// Mitsubishi GX Works2 project: Star delta new1   PLC: FX1S

PROGRAM MAIN
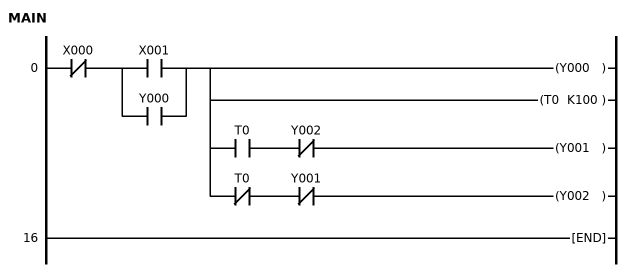
0     LDI     X000
      LD      X001
      OR      Y000
      ANB
      OUT     Y000
      OUT     T0 K100
      MPS
      AND     T0
      ANI     Y002
      OUT     Y001
      MPP
      ANI     T0
      ANI     Y001
      OUT     Y002
16    END
END_PROGRAM
